// TIA Portal V20 export
FUNCTION_BLOCK "FB_DigitalInputsBW_Station"   // FB214, SCL
{ S7_Optimized_Access := 'TRUE' }
// stored: AutoNumber false, MemoryReserve 100, SetENOAutomatically false
   VAR
      sUndrilledPartCtrl { S7_SetPoint := 'True'} : "FB_DigitalInput";
      sDrilledPartCtrl { S7_SetPoint := 'True'} : "FB_DigitalInput";
      sBwCtrl { S7_SetPoint := 'True'} : "FB_DigitalInput";
   END_VAR
BEGIN
   REGION Description head
       //==================================================================================
       // POSALUX Swiss SA / (C) Copyright 2025
       //----------------------------------------------------------------------------------
       // Title: Digital Inputs mapping
       // Comment/Function: BW Station Digital Inputs mapping
       // Author: Fabien WALDT
       // Engineering: TIA Portal v17
       //----------------------------------------------------------------------------------
       // Change log table:
       // Version  | Date     | Expert in charge | Changes applied
       // ---------|----------|------------------|-----------------------------------------
       // 00.00.01 | 20250423 | WFA              | First released version
       // =================================================================================
   END_REGION


   REGION Backwall Station 
       IF "DB_WAF".CtrlInEnable OR "DB_WAF".CtrlOutEnable THEN
           #sUndrilledPartCtrl(iHWStatus := "DB_BwLoaderExchange".Inputs.UndrilledPartControl);
       END_IF;
       IF "DB_WAF".CtrlInEnable OR "DB_WAF".CtrlOutEnable THEN
           #sDrilledPartCtrl(iHWStatus := "DB_BwLoaderExchange".Inputs.DrilledPartControl);
       END_IF;
       IF "DB_WAF".CtrlBwEnable THEN
           #sBwCtrl(iHWStatus := "DB_BwLoaderExchange".Inputs.BackwallControl);
       END_IF;
   END_REGION
END_FUNCTION_BLOCK
